VAR_GLOBAL
////////////////////////////////////////:	///////////////////////////////////////////////////
/////////////////////////////////////////////////////////////////////////////////////GENERIC/////////////////////////////////////////////////////////////////////////////////////

	stHMI_IO							: ST_HMI_IO;
	bQuitHMI							: BOOL;
	bShutDown							: BOOL;
	stStatusBanner						: ST_StatusBanner;
	nPopUp								: DINT;
	stTableCycleDataNest1				: ARRAY[0..2000] OF ST_TableCycleData;
	stTableCycleDataNest2				: ARRAY[0..2000] OF ST_TableCycleData;
	
	

/////////////////////////////////////////////////////////////////////////////////////SYSTEM INFO/////////////////////////////////////////////////////////////////////////////////////

	sSoftwareVersion					: STRING := ' 1.0 ';
	sSoftwareDate						: STRING := ' 10.December.2024 ';
	sTC3Version							: STRING := ' v3.1.4024.53, Runtime v3.1.4024.40 ';
	sHMIVersion							: STRING := ' TcXaeShell Version 15.0.28010.2050 D15.8 ';
	sSystemName							: STRING := ' Print & Applay Labeller ' ;
	sProjectID							: STRING := ' TE 1099 PAL' ;
	sAplication                     	: STRING := ' Print & Applay Labeller ';
	sHMIServer                			: STRING := ' ---- ';
	
	NetAmsId        	       			: T_AmsNetId := '192.168.7.20.1.1'; // AMS-ID for com port setup 
	
/////////////////////////////////////////////////////////////////////////////////////USER LOG/////////////////////////////////////////////////////////////////////////////////////

	sUserGroupIn						: STRING;
	sUserGroupOut						: STRING;
	sUserName							: STRING;
	bUserLoggedIn						: BOOL;			
	bLogOut								: BOOL;	
	rUserLoggedIn						: R_TRIG;

/////////////////////////////////////////////////////////////////////////////////////MANUAL/////////////////////////////////////////////////////////////////////////////////////

	bEnableManual						: BOOL;
	nMainRegion							: DINT;
	bManualModeOffFlag					: BOOL;
	

	
	
	stAnimations						: ST_Animations;
	nMachineDefinitionIndex				: INT;
	bMachineDefinitionSet				: BOOL;
	
	bProcessCylinder1_Up				: BOOL;
	bProcessCylinder1_Down				: BOOL;
	bProcessCylinder2_Up				: BOOL;
	bProcessCylinder2_Down				: BOOL;
	
	bProcessDoor_Up						: BOOL;
	bProcessDoor_Down					: BOOL;
	
	bLeaktester1_Start					: BOOL;
	bLeaktester2_Start					: BOOL;
	bLeaktester1_Stop					: BOOL;
	bLeaktester2_Stop					: BOOL;
	bLeaktester1_Reset					: BOOL;
	bLeaktester2_Reset					: BOOL;
	bCameraResetStatistics				: ARRAY[1..4] OF BOOL;
	bCameraSettingNo					: ARRAY[1..4] OF UINT;
	bCameraSettingVal					: ARRAY[1..4] OF UDINT;
	bCameraSetTreshold					: ARRAY[1..4] OF BOOL;
	bCameraTrigger						: ARRAY[1..4] OF BOOL;
	
	//Probes
	bSetTolerances						: BOOL;
	abPresetProbe						: ARRAY [1..8] OF BOOL;
	bSetCalibrationBlock1				: BOOL;
	bSetCalibrationBlock2				: BOOL;
	bEnableSetCablibrationBlock1		: BOOL;
	bEnableSetCablibrationBlock2		: BOOL;
	bSetDistances						: BOOL;
	
	
	
	
/////////////////////////////////////////////////////////////////////////////////////Generics/////////////////////////////////////////////////////////////////////////////////////	
		
	bLeftHand							: BOOL;
	bRightHand							: BOOL;
	
END_VAR

VAR_GLOBAL PERSISTENT
	
	stTimers							: ST_Timers;
	stStatisticsHMI						: ARRAY [0..6] OF ST_StatisticsHMI;	//0: GENERAL
																	//1: Leak Tester 1
																	//2: Leak Tester 2
																	//3: Height Test 1
																	//4: Height Test 2
																	//5: Camera set 1
																	//6: camera set 2
														
	/////////////////////////////////////////////////////////////////////////////////////SETTINGS/////////////////////////////////////////////////////////////////////////////////////	
	


	
	//TwinSAFE
	
	nAirPressureMaxValue				: UINT;	
	nAirPressureMinValue				: UINT;	
	abMachineDefinition					: ARRAY[1..5] OF  BOOL;
	

	

	
END_VAR

(* stored: Version 1.1.0.1, ProductVersion 3.1.4026.17
   GVL GVL_HMI: Id {7d424ba3-5d42-48e0-870b-7d749b127bab} *)
